// SIMATIC S7-200 project (STEP 7-Micro/WIN), CPU 224XP CN REL 02.01

SYMBOL_TABLE 用户定义1
Auto_Manual      V0.0     // 自动
G_num            VW220    // 关计数
K_num            VW200    // 开计数
JSQL             V1.0     // 计数清零
Gstop            Q0.3     // 关停止
Gout             Q0.2     // 关输出
Kstop            Q0.1     // 开停止
Kout             Q0.0     // 开输出
GTTime           VW112    // 关停止时间
GTime            VW108    // 关延时间
KTTime           VW104    // 开后停止时间
KTime            VW100    // 开延时时间
END_SYMBOL_TABLE

ORGANIZATION_BLOCK 主程序:OB1
TITLE=程序注释
BEGIN
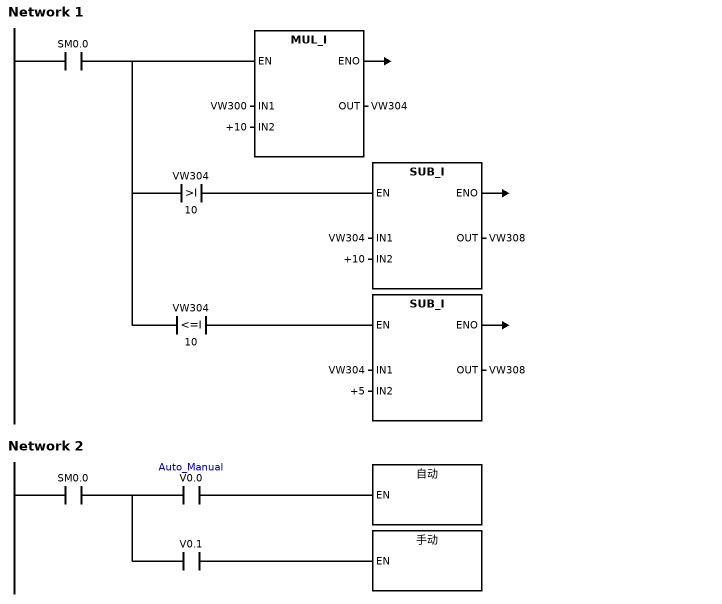
Network 1
LD     SM0.0
LPS
MOVW   VW300, VW304
*I     +10, VW304
AW>    VW304, 10
MOVW   VW304, VW308
-I     +10, VW308
LPP
AW<=   VW304, 10
MOVW   VW304, VW308
-I     +5, VW308
Network 2
LD     SM0.0
LPS
A      Auto_Manual:V0.0
CALL   自动:SBR0
LPP
A      V0.1
CALL   手动:SBR1
END_ORGANIZATION_BLOCK

SUBROUTINE_BLOCK 自动:SBR0
TITLE=子程序注释
BEGIN
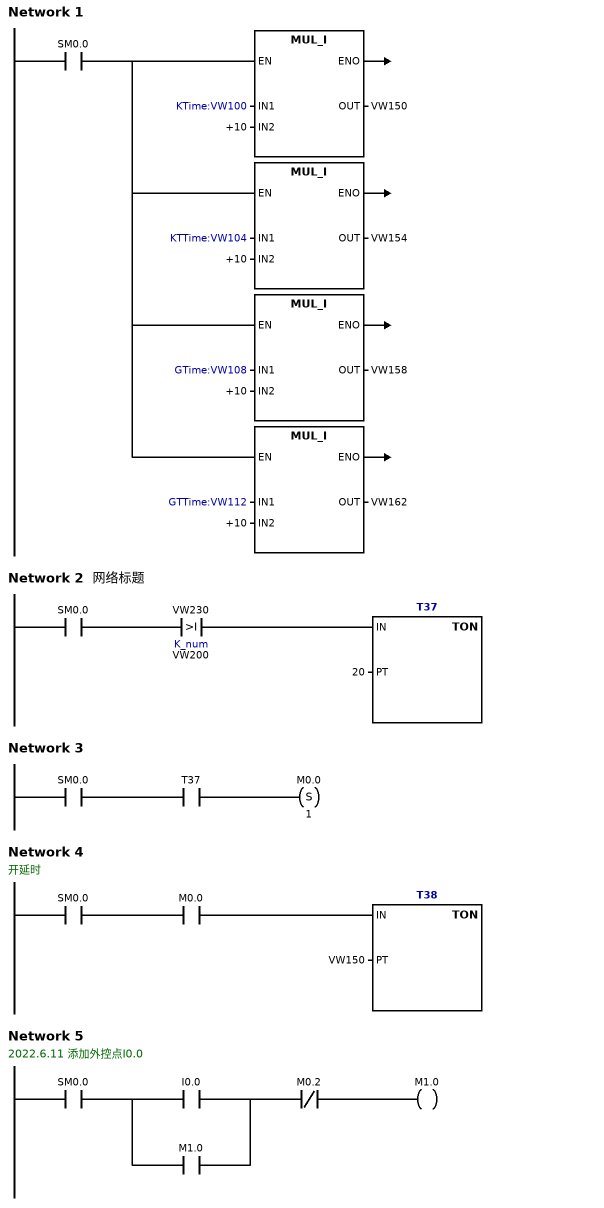
Network 1
LD     SM0.0
MOVW   KTime:VW100, VW150
*I     +10, VW150
MOVW   KTTime:VW104, VW154
*I     +10, VW154
MOVW   GTime:VW108, VW158
*I     +10, VW158
MOVW   GTTime:VW112, VW162
*I     +10, VW162
Network 2 // 网络标题
LD     SM0.0
AW>    VW230, K_num:VW200
TON    T37, 20
Network 3
LD     SM0.0
A      T37
S      M0.0, 1
Network 4
// 开延时
LD     SM0.0
A      M0.0
TON    T38, VW150
Network 5
// 2022.6.11 添加外控点I0.0
LD     SM0.0
LD     I0.0
O      M1.0
ALD
AN     M0.2
=      M1.0
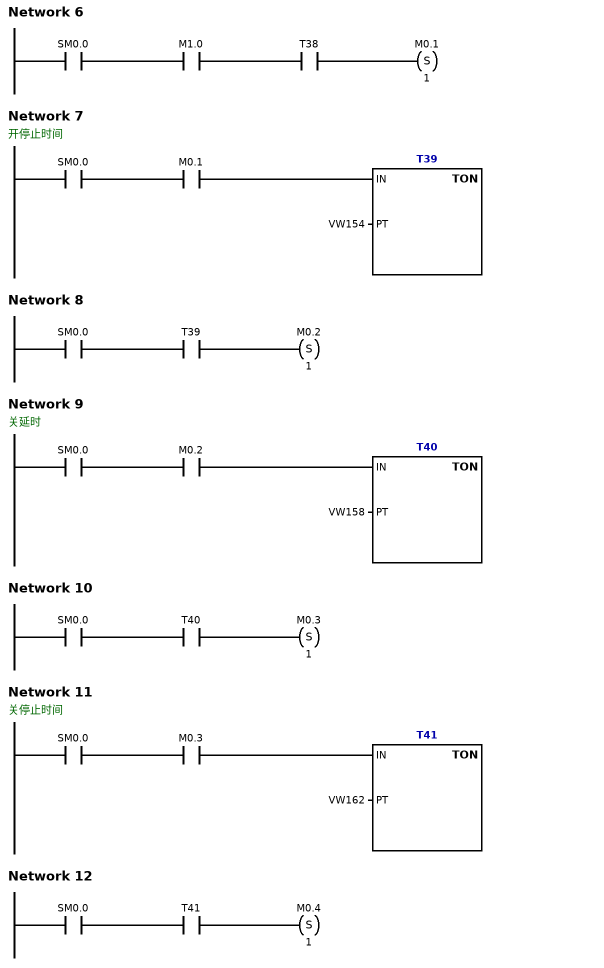
Network 6
LD     SM0.0
A      M1.0
A      T38
S      M0.1, 1
Network 7
// 开停止时间
LD     SM0.0
A      M0.1
TON    T39, VW154
Network 8
LD     SM0.0
A      T39
S      M0.2, 1
Network 9
// 关延时
LD     SM0.0
A      M0.2
TON    T40, VW158
Network 10
LD     SM0.0
A      T40
S      M0.3, 1
Network 11
// 关停止时间
LD     SM0.0
A      M0.3
TON    T41, VW162
Network 12
LD     SM0.0
A      T41
S      M0.4, 1
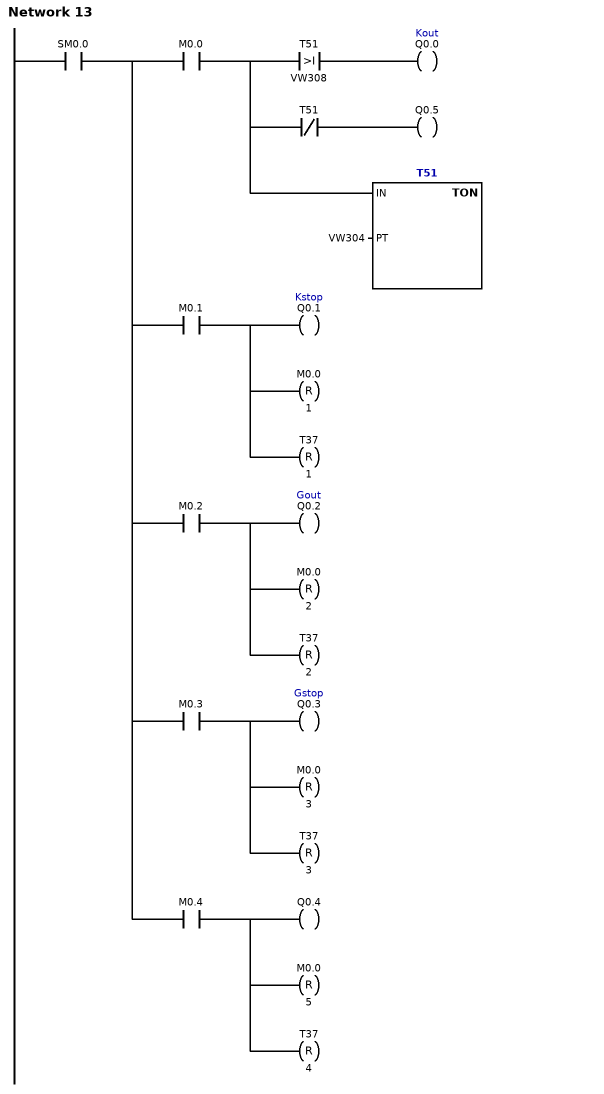
Network 13
LD     SM0.0
LPS
A      M0.0
LPS
AW>    T51, VW308
=      Kout:Q0.0
LRD
AN     T51
=      Q0.5
LPP
TON    T51, VW304
LRD
A      M0.1
=      Kstop:Q0.1
R      M0.0, 1
R      T37, 1
LRD
A      M0.2
=      Gout:Q0.2
R      M0.0, 2
R      T37, 2
LRD
A      M0.3
=      Gstop:Q0.3
R      M0.0, 3
R      T37, 3
LPP
A      M0.4
=      Q0.4
R      M0.0, 5
R      T37, 4
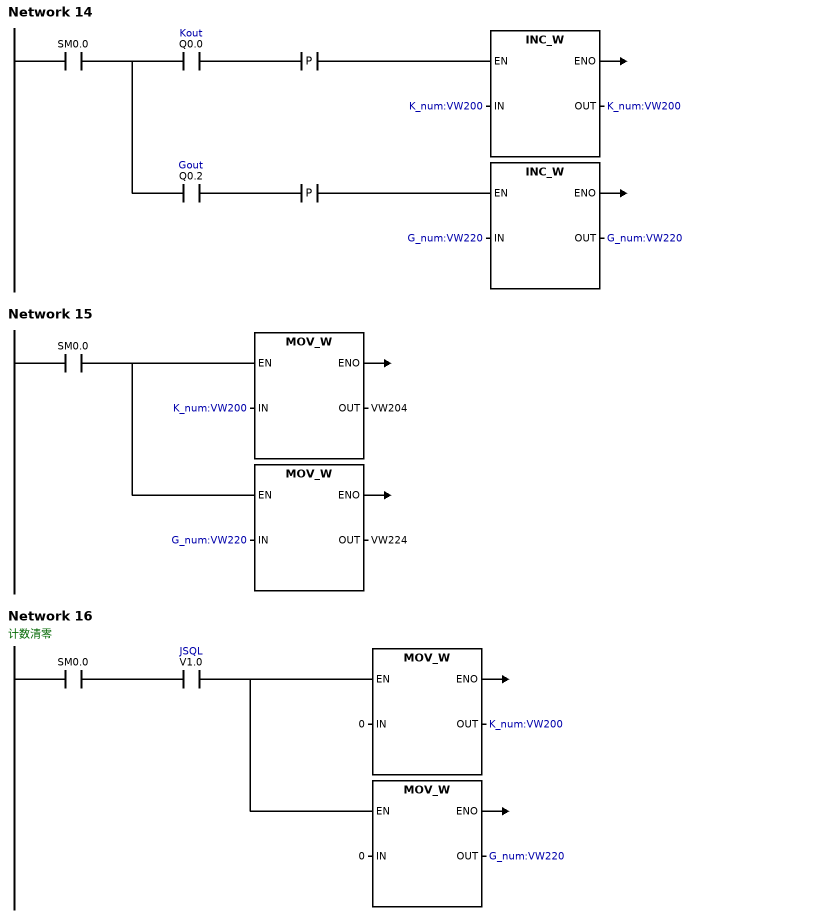
Network 14
LD     SM0.0
LPS
A      Kout:Q0.0
EU
INCW   K_num:VW200
LPP
A      Gout:Q0.2
EU
INCW   G_num:VW220
Network 15
LD     SM0.0
MOVW   K_num:VW200, VW204
MOVW   G_num:VW220, VW224
Network 16
// 计数清零
LD     SM0.0
A      JSQL:V1.0
MOVW   0, K_num:VW200
MOVW   0, G_num:VW220
END_SUBROUTINE_BLOCK

SUBROUTINE_BLOCK 手动:SBR1
TITLE=子程序注释
BEGIN
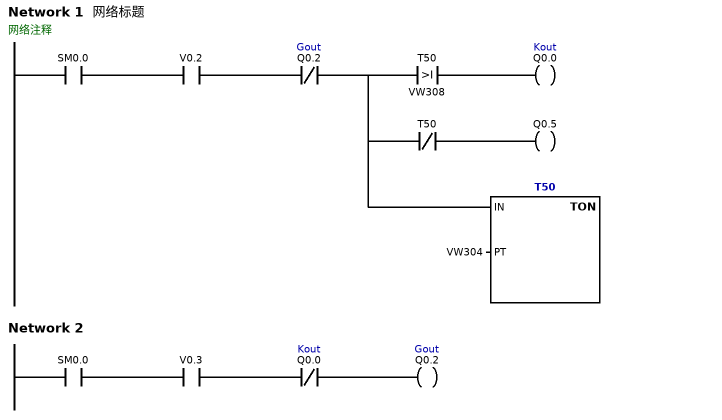
Network 1 // 网络标题
// 网络注释
LD     SM0.0
A      V0.2
AN     Gout:Q0.2
LPS
AW>    T50, VW308
=      Kout:Q0.0
LRD
AN     T50
=      Q0.5
LPP
TON    T50, VW304
Network 2
LD     SM0.0
A      V0.3
AN     Kout:Q0.0
=      Gout:Q0.2
END_SUBROUTINE_BLOCK
